// TIA Portal V20 export
TYPE "zp_CITI_Features"
// stored: Namespace CITI_Logic
   STRUCT
      Map_Enable : Bool;   // Map Enable
      RemoteConfig_En : Bool := FALSE;   // Use Remote Configuration Values
      SL_Enable : Bool := FALSE;   // Map Controls Flashing Green SL
      AndonMap_En : Bool := FALSE;   // Use Map 0 as an Andon Map
      Fault_Data : Bool := FALSE;   // Enable Fault Data Logic
      StringData : Bool := FALSE;   // Map Uses String Data
      Blocked : Bool := FALSE;   // Enable Blocked Logic
      Starved : Bool := FALSE;   // Enable Starved Logic
      Loading : Bool := FALSE;   // Enable Loading Logic
      Unloading : Bool := FALSE;   // Enable Unloading Logic
      Idle : Bool := FALSE;   // Enable Idle Logic
      Wait_1 : Bool := FALSE;   // Enable Wait 1 Logic
      Wait_2 : Bool := FALSE;   // Enable Wait 2 Logic
      Wait_3 : Bool := FALSE;   // Enable Wait 3 Logic
      Wait_4 : Bool := FALSE;   // Enable Wait 4 Logic
      OperatorOvercycle1 : Bool := FALSE;   // Enable Operator Overcycle 1 Logic
      OperatorOvercycle2 : Bool := FALSE;   // Enable Operator Overcycle 2 Logic
      ManualMode : Bool := FALSE;   // Enable Manual Mode Logic
      QualityCheck : Bool := FALSE;   // Enable Quality Check Logic
      ToolChange : Bool := FALSE;   // Enable Tool Change Logic
      MaterialLow : Bool := FALSE;   // Enable Material Low Logic
      EnergyConservation : Bool := FALSE;   // Enable Energy Conservation Logic
      SafetyChecksum : Bool := FALSE;   // Enable Safety Checksum OK Logic
      Bypass : Bool := FALSE;   // Enable Bypass Logic
      Bypass_Cnt : Bool := FALSE;   // Enable Bypass Count
      GoodPart_Cnt : Bool := FALSE;   // Enable Good Part Logic
      RejectPart_Cnt : Bool := FALSE;   // Enable Reject Part Logic
      PUN : Bool := FALSE;   // Map has a PUN
      BufferBypass : Bool := FALSE;   // Enable Buffer Bypass Logic
      PartType : Bool := FALSE;   // Map uses a Part Type
      FTQ : Bool := FALSE;   // Enable FTQ Logic
      AndonHold : Bool := FALSE;   // Enable Andon Hold (Assembly)
      Cycle : Bool := FALSE;   // Enable Cycle Logic
      OnlinePallet_Cnt : Bool := FALSE;   // Enable Online Pallet Counts
      OnlineEmptyPallet_Cnt : Bool := FALSE;   // Enable Online Empty Pallet Counts
      OfflinePallet_Cnt : Bool := FALSE;   // Enable Offline Pallet Counts
      Buffer_Cnt : Bool := FALSE;   // Enable Buffer Count
      PalletID : Bool := FALSE;   // Enable Pallet ID
      ProcessRetry_Cnt : Bool := FALSE;   // Enable Process Retry Counts
      SPC_Cnt : Bool := FALSE;   // Enable SPC Counts
      GM_PN : Bool := FALSE;   // Map Uses GM Part Number
      Opt_Data : Bool := FALSE;   // Map Uses Optional Data
      CMM_Data : Bool := FALSE;   // Enable CMM Data
      "Filter Data" : Bool := FALSE;   // Enable Filter Data
      Tank_Level : Bool := FALSE;   // Enable HPC Tank Level Low
      Pump_Back_Level : Bool := FALSE;   // Enable HPC Pump Back Level Okay
      Tank_Coolant_Temp : Bool := FALSE;   // Enable HPC Tank Coolant Temperature Low
      DryCycle_Mode : Bool := FALSE;   // Enable Dry Cycle Mode
      Using_GCCS_Template : Bool := FALSE;   // Using a GCCS Template
   END_STRUCT;
END_TYPE
